{attribute 'linkalways'} 
{attribute 'no_explicit_call' := 'This FB is a CLASS and must be accessed using methods or properties'}
{attribute 'enable_dynamic_creation'}
FUNCTION_BLOCK _ETcVnInterpolationType EXTENDS EnumDatatypeBase
VAR
	localData : ETcVnInterpolationType;
	activeData : REFERENCE TO ETcVnInterpolationType;
	enumBaseDatatype : _DINT(localData);
END_VAR

METHOD PRIVATE AddLocalEnumeration
VAR_INPUT
	Enumeration : T_MAXSTRING;
	Value : ETcVnInterpolationType;
END_VAR
AddEnumeration(Enumeration, Value);
END_METHOD

PROPERTY PUBLIC Address : PVOID
GET
Address := ADR(activeData);
END_GET
END_PROPERTY

METHOD PUBLIC ClearReference
VAR_INPUT
END_VAR
activeData REF= localData;
SetBaseDatatypeReference();
END_METHOD

METHOD PUBLIC Clone : I_Datatype
VAR
    pClone : POINTER TO _ETcVnInterpolationType;
END_VAR
pClone := __NEW(_ETcVnInterpolationType(InitialValue := Value));
Clone := pClone^;
END_METHOD

METHOD FB_init : BOOL
VAR_INPUT
	bInitRetains : BOOL; // if TRUE, the retain variables are initialized (warm start / cold start)
	bInCopyCode : BOOL;  // if TRUE, the instance afterwards gets moved into the copy code (online change)
	InitialValue : ETcVnInterpolationType;
END_VAR
localData := InitialValue;
AddBaseDatatype(enumBaseDatatype);
ClearReference();

AddLocalEnumeration('TCVN_IT_NEAREST_NEIGHBOR', ETcVnInterpolationType.TCVN_IT_NEAREST_NEIGHBOR);
AddLocalEnumeration('TCVN_IT_BILINEAR', ETcVnInterpolationType.TCVN_IT_BILINEAR);
AddLocalEnumeration('TCVN_IT_BICUBIC', ETcVnInterpolationType.TCVN_IT_BICUBIC);
AddLocalEnumeration('TCVN_IT_AREA_BASED', ETcVnInterpolationType.TCVN_IT_AREA_BASED);
AddLocalEnumeration('TCVN_IT_LANCZOS4', ETcVnInterpolationType.TCVN_IT_LANCZOS4);
END_METHOD

PROPERTY PUBLIC Identifier : T_MAXSTRING
GET
Identifier := 'ETcVnInterpolationType';
END_GET
END_PROPERTY

METHOD IsEnumeratorValueEqual : BOOL
VAR_INPUT
	Enumerator : I_KeyValueForwardEnumerator;
END_VAR
VAR
	storedValue : ETcVnInterpolationType;
END_VAR
IF NOT Enumerator.TryGet(storedValue) THEN
	RETURN;
END_IF

IsEnumeratorValueEqual := storedValue = activeData;
END_METHOD

METHOD PUBLIC MakeReferenceTo
VAR_INPUT
	ReferenceTarget : REFERENCE TO ETcVnInterpolationType;
END_VAR
activeData REF= ReferenceTarget;
SetBaseDatatypeReference();
END_METHOD

METHOD PROTECTED SetBaseDatatypeReference
VAR_INPUT
END_VAR
enumBaseDatatype.MakeReferenceTo(activeData);
END_METHOD

PROPERTY PUBLIC Size : UDINT
GET
Size := SIZEOF(activeData);
END_GET
END_PROPERTY

METHOD TryMakeReferenceTo : BOOL
VAR_INPUT
	Target : I_Datatype;
END_VAR
VAR
	targetAsEnum : I_EnumDatatype;
	pTargetData : POINTER TO ETcVnInterpolationType;
END_VAR
IF NOT Target.TryResolveAsEnumDatatype(targetAsEnum) THEN
	RETURN;
END_IF

IF targetAsEnum.Identifier <> Identifier THEN
	RETURN;
END_IF

pTargetData := Target.Address;
activeData REF= pTargetData^;
SetBaseDatatypeReference();
TryMakeReferenceTo := TRUE;
END_METHOD

PROPERTY PUBLIC Value : ETcVnInterpolationType
GET
Value := activeData;
END_GET
SET
activeData := Value;
END_SET
END_PROPERTY

END_FUNCTION_BLOCK

(* stored: Version 1.1.0.1
   POU _ETcVnInterpolationType: Id {019d4e34-27a1-430f-a214-7449353cc676}, SpecialFunc None
   Folder Constructor: Id {19fc23c2-9062-4ccc-b5a2-7f98ef271b40}
   Folder Private: Id {2d1c4cea-384d-4104-b5a8-aefb4f15ef51}
   Folder Protected: Id {0444251e-07af-4fb1-84da-eae3f7d20a17}
   Method AddLocalEnumeration: Id {7e2f9adc-da99-4f0c-9e27-878cbfbdaa8f}
   Property Address: Id {c9bf2433-2f81-4797-be98-2b56cfd138dc}
   Get Get: Id {6cf79caa-f519-4f55-8c13-b9b06b2063dc}
   Method ClearReference: Id {8c44a6c8-1510-4ba8-b0ab-ed639a216418}
   Method Clone: Id {876b8ea5-872b-4032-8c9e-4cbf4bee10a1}
   Method FB_init: Id {2be5c705-5e2f-4ef1-b49c-cd4603ac23ff}
   Property Identifier: Id {79af02ea-90f6-49e9-9880-6de1035da6b9}
   Get Get: Id {82b081d7-a8f4-4010-8427-9690ec38d3f7}
   Method IsEnumeratorValueEqual: Id {a2d2443c-4e01-46bc-b56d-3f6adb10ea8a}
   Method MakeReferenceTo: Id {e13abcb2-b240-40b5-8665-9b1593fb1c23}
   Method SetBaseDatatypeReference: Id {5cf864ae-bbe9-4902-9644-bcc8c5325c70}
   Property Size: Id {4428a56c-2474-4253-ad87-b7e43e9fdb7f}
   Get Get: Id {f7a1c84f-c1d2-43f5-a322-1dae1c642563}
   Method TryMakeReferenceTo: Id {bb739a99-bde5-49e2-b10b-71d8b44a29e9}
   Property Value: Id {dd29573e-5c94-46b8-a73e-82b1a55773de}
   Get Get: Id {a91f0af8-1071-4a04-83ee-9268dd650111}
   Set Set: Id {04460000-c4c7-4aeb-ba55-8c1b630256bb} *)
